FUNCTION_BLOCK QualityInspectionSequenceAutomatic EXTENDS QualityInspectionSequence IMPLEMENTS ZCore.ISequence
VAR
  _step : ZCore.Step(QualityInspectionStep.AutomaticBegin, QualityInspectionStep.AutomaticEnd);
  _timer : ZAux.Timer;
  _simTimer : ZAux.Timer;
END_VAR

IF NOT Busy THEN
  RETURN;
END_IF

IF OnStart(_step) THEN
  ; // init custom sequence variables here ...
END_IF

IF OnStop() THEN
  RETURN; // external stop was triggered
END_IF

IF OnHalt() THEN
  ; // Halting := TRUE; // Uncomment to acknowledge that the sequence is halting
END_IF

REPEAT
  LogStep();

  CASE _step.Index OF
    (* -------------------------------------------------------------------------------------------------------------------------------- *)
    QualityInspectionStep.AutomaticBegin:
    (* -------------------------------------------------------------------------------------------------------------------------------- *)
      IF _step.OnEntry()
      THEN
        _timer.WaitAsync(1.0);
      END_IF

      _step.SetNext(QualityInspectionStep.AutomaticEnableLight);

    (* -------------------------------------------------------------------------------------------------------------------------------- *)
    QualityInspectionStep.AutomaticEnableLight:
    (* -------------------------------------------------------------------------------------------------------------------------------- *)
      IF _step.OnEntry()
      THEN        
        _io.EnableLight.Enable(TRUE);
      END_IF
      
      _step.SetNext(index:=QualityInspectionStep.AutomaticTriggerCam);

    (* -------------------------------------------------------------------------------------------------------------------------------- *)
    QualityInspectionStep.AutomaticTriggerCam:
    (* -------------------------------------------------------------------------------------------------------------------------------- *)
      IF _step.OnEntry()
      THEN        
        _io.TriggerCam.Duration := 0.5;
        _io.TriggerCam.RunAsync(startToken:=THIS^);
      END_IF
      
      Await(obj1:=_io.TriggerCam, nextStep:=QualityInspectionStep.AutomaticWaitTillCamSendsOk);

    (* -------------------------------------------------------------------------------------------------------------------------------- *)
    QualityInspectionStep.AutomaticWaitTillCamSendsOk:
    (* -------------------------------------------------------------------------------------------------------------------------------- *)
      IF _step.OnEntry()
      THEN        
        _simTimer.WaitAsync(1.5);
      END_IF
      
      IF _simTimer.Done
      THEN
        _io.CamOk.Enable(TRUE);
			END_IF
      
      IF _io.CamOk.RisingTrigger()
      THEN
        _io.CamOk.Enable(FALSE);
        _step.SetNext(index:=QualityInspectionStep.AutomaticEnd);
      END_IF
    
    (* -------------------------------------------------------------------------------------------------------------------------------- *)
    QualityInspectionStep.AutomaticEnd:
    (* -------------------------------------------------------------------------------------------------------------------------------- *)
      SetBusy(FALSE);
  
  ELSE
    Abort('sequence contains unhandled step');
  END_CASE
UNTIL _step.IsNotRepeatable() OR_ELSE NOT Busy END_REPEAT

END_FUNCTION_BLOCK

(* stored: Version 1.1.0.1
   POU QualityInspectionSequenceAutomatic: Id {05c6a32c-1cb2-4aab-a4cc-ce8a269ff3ed}, SpecialFunc None *)
